// TwinCAT 3 PLC project Untitled1
// ProgramVersion: 3.1.4023.0
// libraries:
//   Tc2_MC2, * (Beckhoff Automation GmbH)
//   Tc2_Standard, * (Beckhoff Automation GmbH)
//   Tc2_System, * (Beckhoff Automation GmbH)
//   Tc2_Utilities, * (Beckhoff Automation GmbH)
//   Tc3_Module, * (Beckhoff Automation GmbH)
// project tree:
//   DUTs/ A21ToolStorage.TcDUT (not stored), Bundle.TcDUT (not stored), EOAT.TcDUT (not stored), Interval.TcDUT (not stored), ONE_BIT.TcDUT (not stored), PositionMaterials.TcDUT (not stored)
//   DUTs/Enums/ A21.TcDUT (not stored), Chipboard.TcDUT (not stored), Homing.TcDUT (not stored), SectionEnum.TcDUT (not stored), Surface.TcDUT (not stored), WoodBunk.TcDUT (not stored)
//   DUTs/Insertion/Drives/ AirPiston.TcPOU (not stored), ClearLinkMC.TcPOU, SimplePiston.TcPOU (not stored)
//   DUTs/Insertion/ Insertion.TcPOU, SuctionPad.TcDUT (not stored)
//   DUTs/Insertion/Prototypes/ FBA_Drive.TcPOU, I_ContinuousDrive.TcIO (not stored), I_Drive.TcIO, I_PositionalDrive.TcIO (not stored), I_EncodedDrive.TcIO (not stored)
//   DUTs/Machines/ KukaRobot.TcPOU, RobotA21.TcPOU, StrapMachine.TcPOU
//   DUTs/Material Holders/ SkidMagazine.TcPOU, MaterialHolder.TcPOU, WoodBunkTable.TcPOU
//   GVLs/ GVL.TcGVL (not stored), Hardware.TcGVL
//   / PlcTask.TcTTO
//   POUs/ MAIN.TcPOU
//   POUs/Module Calls/ CallHardwareModules.TcPOU, SetSuctions.TcPOU (not stored), SetupHardware.TcPOU
//   POUs/Utility/ BoolArrayToInteger.TcPOU, CEILING.TcPOU (not stored), IntegerBitAccess.TcPOU (not stored), IntegerToBoolArray.TcPOU (not stored), JoinStrings.TcPOU (not stored), WithinTolerance.TcPOU (not stored)
//   POUs/Utility/String Array/ AddToStringArray.TcPOU, RemoveElementFromStringArray.TcPOU (not stored), RemoveIndexFromStringArray.TcPOU (not stored), StringArrayCloseGaps.TcPOU (not stored)
// real-time tasks:
//   TASK PlcTask: cycle T#10ms, priority 20, ADS port 350
// I/O:
//   DEVICE Device 1 (EtherCAT), AmsNetId 5.131.216.41.2.1
//     EK1200 [EK1200-5000 EtherCAT Power supply (2A E-Bus)]
//       IPC_O [EL2809 16Ch. Dig. Output 24V, 0.5A]
//       JUNC_A21 [EK1122 2 port EtherCAT junction]
//         C4 [EK1100 EtherCAT Coupler (2A E-Bus)]
//           C4_I1 [EL1809 16Ch. Dig. Input 24V, 3ms]
//           C4_O2 [EL2809 16Ch. Dig. Output 24V, 0.5A]
//           C4_O3 [EL2809 16Ch. Dig. Output 24V, 0.5A]
//           BRIDGE_ROBOT1 [EL6695 EtherCAT Bridge terminal (Primary)]
//           Term 14 (EL9011) [EL9011 End Terminal]
//         SB01 [EP1809-0021 16 Ch. Dig. Input 24V, 3ms, M8]
//         SB05 [EP1008-0001 8 Ch. Dig. Input 24V, 3ms, M8]
//         SB04 [EP1809-0021 16 Ch. Dig. Input 24V, 3ms, M8]
//         SB03 [EP1008-0001 8 Ch. Dig. Input 24V, 3ms, M8]
//         C1 [EK1100 EtherCAT Coupler (2A E-Bus)]
//           C1_I1 [EL1809 16Ch. Dig. Input 24V, 3ms]
//           C1_O2 [EL2809 16Ch. Dig. Output 24V, 0.5A]
//           BRIDGE_ROBOT2 [EL6695 EtherCAT Bridge terminal (Primary)]
//           Term 13 (EL9011) [EL9011 End Terminal]
//         SB02 [EP1809-0021 16 Ch. Dig. Input 24V, 3ms, M8]
//         SB07 [EP1008-0001 8 Ch. Dig. Input 24V, 3ms, M8]
//         SB06 [EP1008-0001 8 Ch. Dig. Input 24V, 3ms, M8]
// variable links:
//   Untitled1/Untitled1 Instance <-> Device 1 (EtherCAT)/EK1200/JUNC_A21/C1/BRIDGE_ROBOT2
//     PlcTask Inputs/Hardware.robotRight.inputs[{2..20}] <-> IO Inputs/In_{2..20}  (19 links)
//     PlcTask Inputs/Hardware.robotRight.inputs[1] <-> IO Inputs/In
//     PlcTask Outputs/Hardware.robotRight.outputs[{2..50}] <-> IO Outputs/Out_{2..50}  (49 links)
//     PlcTask Outputs/Hardware.robotRight.outputs[1] <-> IO Outputs/Out
//   Untitled1/Untitled1 Instance <-> Device 1 (EtherCAT)/EK1200/JUNC_A21/C1/C1_I1
//     PlcTask Inputs/Hardware.strapper.done <-> Channel 4/Input
//     PlcTask Inputs/Hardware.strapper.error <-> Channel 1/Input
//     PlcTask Inputs/Hardware.strapper.home <-> Channel 5/Input
//     PlcTask Inputs/Hardware.strapper.ready <-> Channel 2/Input
//   Untitled1/Untitled1 Instance <-> Device 1 (EtherCAT)/EK1200/JUNC_A21/C1/C1_O2
//     PlcTask Outputs/Hardware.strapper.enable <-> Channel 2/Output
//     PlcTask Outputs/Hardware.strapper.execute <-> Channel 1/Output
//     PlcTask Outputs/Hardware.strapper.reset <-> Channel 3/Output
//   Untitled1/Untitled1 Instance <-> Device 1 (EtherCAT)/EK1200/JUNC_A21/C4/BRIDGE_ROBOT1
//     PlcTask Inputs/Hardware.robotLeft.inputs[{2..20}] <-> IO Inputs/In_{2..20}  (19 links)
//     PlcTask Inputs/Hardware.robotLeft.inputs[1] <-> IO Inputs/In
//     PlcTask Outputs/Hardware.robotLeft.outputs[{2..50}] <-> IO Outputs/Out_{2..50}  (49 links)
//     PlcTask Outputs/Hardware.robotLeft.outputs[1] <-> IO Outputs/Out
//   Untitled1/Untitled1 Instance <-> Device 1 (EtherCAT)/EK1200/JUNC_A21/C4/C4_I1
//     PlcTask Inputs/Hardware.topSuction[1].occupied <-> Channel 9/Input
//     PlcTask Inputs/Hardware.topSuction[2].occupied <-> Channel 10/Input
//     PlcTask Inputs/Hardware.topSuction[3].occupied <-> Channel 11/Input
//     PlcTask Inputs/Hardware.verticalDriveLeft.home <-> Channel 3/Input
//     PlcTask Inputs/Hardware.verticalDriveLeft.innerLimit <-> Channel 2/Input
//     PlcTask Inputs/Hardware.verticalDriveLeft.outerLimit <-> Channel 1/Input
//     PlcTask Inputs/Hardware.verticalDriveRight.home <-> Channel 7/Input
//     PlcTask Inputs/Hardware.verticalDriveRight.innerLimit <-> Channel 6/Input
//     PlcTask Inputs/Hardware.verticalDriveRight.outerLimit <-> Channel 5/Input
//   Untitled1/Untitled1 Instance <-> Device 1 (EtherCAT)/EK1200/JUNC_A21/C4/C4_O2
//     PlcTask Outputs/Hardware.horizontalDriveLeft.valveExtend <-> Channel 5/Output
//     PlcTask Outputs/Hardware.horizontalDriveLeft.valveRetract <-> Channel 6/Output
//     PlcTask Outputs/Hardware.horizontalDriveRight.valveExtend <-> Channel 15/Output
//     PlcTask Outputs/Hardware.horizontalDriveRight.valveRetract <-> Channel 16/Output
//     PlcTask Outputs/Hardware.leftSuction[{1..4}].enable <-> Channel {7..10}/Output  (4 links)
//     PlcTask Outputs/Hardware.verticalDriveLeft.brakeRelease <-> Channel 4/Output
//     PlcTask Outputs/Hardware.verticalDriveRight.brakeRelease <-> Channel 14/Output
//   Untitled1/Untitled1 Instance <-> Device 1 (EtherCAT)/EK1200/JUNC_A21/C4/C4_O3
//     PlcTask Outputs/Hardware.bottomSuction[1].enable <-> Channel 7/Output
//     PlcTask Outputs/Hardware.bottomSuction[2].enable <-> Channel 8/Output
//     PlcTask Outputs/Hardware.pistonBottom.pistonExtend <-> Channel 5/Output
//     PlcTask Outputs/Hardware.pistonBottom.pistonRetract <-> Channel 6/Output
//     PlcTask Outputs/Hardware.rightSuction[{1..4}].enable <-> Channel {1..4}/Output  (4 links)
//     PlcTask Outputs/Hardware.topSuction[1].enable <-> Channel 9/Output
//     PlcTask Outputs/Hardware.topSuction[2].enable <-> Channel 10/Output
//     PlcTask Outputs/Hardware.topSuction[3].enable <-> Channel 11/Output
//   Untitled1/Untitled1 Instance <-> Device 1 (EtherCAT)/EK1200/JUNC_A21/SB01
//     PlcTask Inputs/Hardware.horizontalDriveLeft.home <-> Channel 11/Input
//     PlcTask Inputs/Hardware.horizontalDriveLeft.innerLimit <-> Channel 12/Input
//     PlcTask Inputs/Hardware.leftSuction[{1..4}].occupied <-> Channel {13..16}/Input  (4 links)
//     PlcTask Inputs/Hardware.stagingTableLeft.occupied[{1..10}] <-> Channel {1..10}/Input  (10 links)
//   Untitled1/Untitled1 Instance <-> Device 1 (EtherCAT)/EK1200/JUNC_A21/SB02
//     PlcTask Inputs/Hardware.horizontalDriveRight.home <-> Channel 11/Input
//     PlcTask Inputs/Hardware.horizontalDriveRight.innerLimit <-> Channel 12/Input
//     PlcTask Inputs/Hardware.rightSuction[{1..4}].occupied <-> Channel {13..16}/Input  (4 links)
//     PlcTask Inputs/Hardware.stagingTableRight.occupied[{1..10}] <-> Channel {1..10}/Input  (10 links)
//   Untitled1/Untitled1 Instance <-> Device 1 (EtherCAT)/EK1200/JUNC_A21/SB05
//     PlcTask Inputs/Hardware.magazineLeft.inPosition1 <-> Channel 1/Input
//     PlcTask Inputs/Hardware.magazineLeft.inPosition2 <-> Channel 2/Input
//     PlcTask Inputs/Hardware.skidLeft.inPosition1 <-> Channel 3/Input
//     PlcTask Inputs/Hardware.skidLeft.inPosition2 <-> Channel 4/Input
//   Untitled1/Untitled1 Instance <-> Device 1 (EtherCAT)/EK1200/JUNC_A21/SB06
//     PlcTask Inputs/Hardware.magazineRight.inPosition1 <-> Channel 1/Input
//     PlcTask Inputs/Hardware.magazineRight.inPosition2 <-> Channel 2/Input
//     PlcTask Inputs/Hardware.skidRight.inPosition1 <-> Channel 3/Input
//     PlcTask Inputs/Hardware.skidRight.inPosition2 <-> Channel 4/Input
//   Untitled1/Untitled1 Instance <-> Device 1 (EtherCAT)/EK1200/JUNC_A21/SB07
//     PlcTask Inputs/Hardware.bottomSuction[1].occupied <-> Channel 6/Input
//     PlcTask Inputs/Hardware.bottomSuction[2].occupied <-> Channel 7/Input
//     PlcTask Inputs/Hardware.pistonBottom.extended <-> Channel 5/Input
//     PlcTask Inputs/Hardware.pistonBottom.retracted <-> Channel 4/Input

CONFIGURATION Untitled1
    RESOURCE PLC ON TwinCAT3
        TASK PlcTask(INTERVAL := T#10ms, PRIORITY := 20);
        PROGRAM MAIN WITH PlcTask : MAIN;
    END_RESOURCE
END_CONFIGURATION

// ---- GVLs/Hardware.TcGVL
//{attribute 'qualified_only'}
VAR_GLOBAL
	robotLeft, robotRight : RobotA21;
	toolStorageLeft, toolStorageRight : A21ToolStorage;
	
	skidLeft, skidRight : SkidMagazine;
	
	stagingTableLeft, stagingTableRight : WoodBunkTable;
	magazineLeft, magazineRight : SkidMagazine;
	
	strapper : StrapMachine;
	
	horizontalDriveLeft, horizontalDriveRight : AirPiston;
	verticalDriveLeft, verticalDriveRight : ClearLinkMC;
	pistonBottom : SimplePiston;
	
	topSuction : ARRAY[1..3] OF SuctionPad;
	leftSuction : ARRAY[1..4] OF SuctionPad;
	rightSuction : ARRAY[1..4] OF SuctionPad; 
	bottomSuction : ARRAY[1..2] OF SuctionPad;
END_VAR

// ---- DUTs/Insertion/Prototypes/I_Drive.TcIO
INTERFACE I_Drive

PROPERTY ABSTRACT AtHome : BOOL
GET
END_GET
END_PROPERTY

PROPERTY ABSTRACT AtInnerLimit : BOOL
GET
END_GET
END_PROPERTY

PROPERTY ABSTRACT AtOuterLimit : BOOL
GET
END_GET
END_PROPERTY

PROPERTY ABSTRACT Busy : BOOL
GET
END_GET
END_PROPERTY

PROPERTY ABSTRACT Contact : BOOL
GET
END_GET
END_PROPERTY

PROPERTY ABSTRACT Error : BOOL
GET
END_GET
END_PROPERTY

PROPERTY ABSTRACT HomeSet : BOOL
GET
END_GET
END_PROPERTY

METHOD ABSTRACT homingSequence : BOOL
VAR_INPUT
END_VAR
END_METHOD

METHOD ABSTRACT stop : BOOL
VAR_INPUT
END_VAR
END_METHOD

END_INTERFACE

// ---- POUs/MAIN.TcPOU
PROGRAM MAIN
VAR
	execute : BOOL;
	stop : BOOL;
	generalError : BOOL;
	failLeft, failRight : BOOL;
	
	manualStep : BOOL := TRUE;
	manualSuction : BOOL := FALSE;
END_VAR
VAR //local types
	woodBunkArr : ARRAY[0..GVL.maxPairs] OF PositionMaterials;
	
	stagingTemplateLeft, stagingTemplateRight AT %M* : WoodBunkTable; //declaration with %M* overwrites addresses of local attributes
	stagingArrayLeft, stagingArrayRight : ARRAY[0..GVL.maxPairs*2] OF STRING;
	insertionLeft, insertionRight : Insertion;
END_VAR
VAR //for testing, to be removed when replaced with pressure sensors
	latchLeft, latchRight : BOOL; //prevents SMC sliders from overshooting the inner limit sensor
	
	suctionEnableTop : BOOL;
	suctionEnableLeft : BOOL;
	suctionEnableRight : BOOL;
	suctionEnableBottom : BOOL;
	
	done : BOOL;
	
	demoPairWB : PositionMaterials := (
		position := 0,
		top := 'WDS20',
		left := 'WDS20',
		right := 'WDS20',
		bottom := 'WDS14');
		
	demoPairCIP : PositionMaterials := (
		position := 0,
		top := 'CIP54',
		bottom := 'CIP18');
	
	demoHeight : REAL := 600; //mm
END_VAR
VAR
	robotLeftOutputs, robotRightOutputs : ARRAY[1..11] OF INT;
	
	insertionMaterials : ARRAY[Surface.TOP..Surface.BOTTOM] OF STRING;
	//robotLeftMaterial, robotRightMaterial : STRING;
	
	topSuctionDelay : TON;
	
	step : (IDLE, LOAD_CIP, STAGING, LOAD_WB, PUSH, STRAP, RELEASE, COMPLETE := 1050);
	
	//these 2 ints should replace the 4 ints after
	commandSet : INT;
	commandStepLeft, commandStepRight : INT;
	
	loadSet : INT;
	loadStepLeft, loadStepRight : INT;
	
	stageSet : INT;	
	stageStepLeft, stageStepRight : INT;
	iSlotLeft, iSlotRight : INT(1..10);
END_VAR
VAR //CONSTANT
	sectionID : SectionEnum := SectionEnum.CHIPBOARD;
	idleRobotOutput : ARRAY[1..11] OF INT;
END_VAR

SetupHardware();
CallHardwareModules();
callLocalModules();

woodBunkArr[0] := demoPairWB;

IF stop THEN //may need to turn off suction
	insertionLeft.stop();
	insertionRight.stop();
	pistonBottom.stop();
	
	robotLeft.clearCommand();
	robotRight.clearCommand();
	RETURN;
END_IF


IF NOT (insertionLeft.screw.HomeSet AND insertionRight.screw.HomeSet) THEN
	insertionLeft.homingSequence();
	insertionRight.homingSequence();
	pistonBottom.retract();
	RETURN;
END_IF


CASE step OF
	IDLE:
		IF execute THEN
			execute := FALSE;
			suctionEnableTop := suctionEnableLeft := suctionEnableRight := suctionEnableBottom := FALSE;
			step := STAGING;
		END_IF
		
		SetSuctions(topSuction, suctionEnableTop);
		SetSuctions(leftSuction, suctionEnableLeft);
		SetSuctions(rightSuction, suctionEnableRight);
		SetSuctions(bottomSuction, suctionEnableBottom);
		
	LOAD_CIP:
		IF NOT done THEN
			done := loadCIP(pair:= demoPairWB, error => generalError);
		END_IF
		
		IF
			(manualStep AND_THEN execute) OR
			(NOT manualStep AND_THEN done)
		THEN
			done := FALSE;
			execute := FALSE;
			
			step := STAGING;
		END_IF
		
	STAGING:
		IF NOT done THEN
			done := stage(error => generalError);
		END_IF
		
		IF
			(manualStep AND_THEN execute) OR
			(NOT manualStep AND_THEN done)
		THEN
			execute := FALSE;
			done := FALSE;
			step := LOAD_WB;
		END_IF
	
	LOAD_WB:
		IF NOT done THEN
			done := loadWB(pair := demoPairWB, error => generalError);
		END_IF
		
		IF manualSuction THEN
			SetSuctions(topSuction, suctionEnableTop);
			SetSuctions(leftSuction, suctionEnableLeft);
			SetSuctions(rightSuction, suctionEnableRight);
			SetSuctions(bottomSuction, suctionEnableBottom);
		END_IF
		
		IF
			(manualStep AND_THEN execute) OR
			(NOT manualStep AND_THEN done)
		THEN
			done := FALSE;
			suctionEnableTop := suctionEnableLeft := suctionEnableRight := suctionEnableBottom := FALSE;
			execute := FALSE;
			
			step := PUSH;
		END_IF
		
	PUSH:
		(*
		IF 
			insertionLeft.sliderPos <> demoHeight/2 //OR 
			//insertionRight.sliderPos <> demoHeight/2 //OR 
			//NOT insertionBottom.contact
		THEN
			insertionLeft.slideAbsolute(demoHeight/2);
			//insertionRight.slideAbsolute(demoHeight/2);
			RETURN;
		END_IF
		*)
		
		IF insertionLeft.screw.AtInnerLimit THEN
			latchLeft := TRUE;
		ELSIF NOT latchLeft THEN
			insertionLeft.press();
		END_IF
		
		IF insertionRight.screw.AtInnerLimit THEN
			latchRight := TRUE;
		ELSIF NOT latchRight THEN
			insertionRight.press();
		END_IF
		pistonBottom.extend();
		
		IF
			(manualStep AND_THEN execute) OR
			(latchLeft AND latchRight (*AND insertionBottom.extended*))
		THEN
			latchLeft := latchRight := FALSE;
			execute := FALSE;
			step := STRAP;
		END_IF
		
	STRAP:
		topSuctionDelay(IN:= , PT:= T#1S, Q=> , ET=> );
		
		strapper.bEnable := TRUE;
		IF strapper.done THEN
			topSuctionDelay.IN := FALSE;
			step := RELEASE;
			RETURN;
		END_IF
		
		IF topSuctionDelay.Q THEN
			SetSuctions(topSuction, FALSE);
			SetSuctions(leftSuction, FALSE);
			SetSuctions(rightSuction, FALSE);
			SetSuctions(bottomSuction, FALSE);
		ELSIF strapper.atBundleLevel THEN
			topSuctionDelay.IN := TRUE;
		END_IF
		
		IF strapper.ready THEN
			strapper.strap();
		END_IF
		
		IF execute THEN
			topSuctionDelay.IN := FALSE;
			execute := FALSE;
			step := RELEASE;
		END_IF
		
	RELEASE: //release command		
		//insertionLeft.slideAbsolute(0);
		//insertionRight.slideAbsolute(0);
		
		insertionLeft.release();
		insertionRight.release();
		pistonBottom.retract();
		
		IF 
			(insertionLeft.screw.AtHome AND insertionRight.screw.AtHome AND pistonBottom.retracted) OR
			execute
		THEN
			execute := FALSE;
			step := COMPLETE;
		END_IF
	
	COMPLETE:
		//reset everything
		step := IDLE;
		
END_CASE

CallHardwareModules(); //end program with hardware call

METHOD callLocalModules : BOOL
stagingTemplateLeft();
stagingTemplateRight();

insertionLeft(
	enable:= TRUE, 
	slider:= verticalDriveLeft, 
	screw:= horizontalDriveLeft, 
	contact=> , 
	softContact=> , 
	busy=> , 
	error=> , 
	home=> , 
	homingComplete=> , 
	sliderPos=> );
	
insertionRight(
	enable:= TRUE, 
	slider:= verticalDriveRight, 
	screw:= horizontalDriveRight,  
	contact=> , 
	softContact=> , 
	busy=> , 
	error=> , 
	home=> , 
	homingComplete=> , 
	sliderPos=> );
END_METHOD

METHOD changeRobotsEOAT : BOOL
VAR_IN_OUT
	robot : RobotA21;
END_VAR
VAR_INPUT
	targetTool : SectionEnum;
END_VAR
IF robotLeft.tool <> targetTool THEN
	MEMSET(ADR(robotLeftOutputs), 0, SIZEOF(robotLeftOutputs));
	
	CASE targetTool OF
		SectionEnum.CHIPBOARD: robotLeftOutputs[1] := A21.TOOL_CHANGE_CHIPBOARD;
		SectionEnum.WOOD_BUNK: robotLeftOutputs[1] := A21.TOOL_CHANGE_BUNK;
	END_CASE
	
	robotLeft.setCommand(robotLeftOutputs);
END_IF

IF robotRight.tool <> targetTool THEN
	MEMSET(ADR(robotRightOutputs), 0, SIZEOF(robotRightOutputs));
	
	CASE targetTool OF
		SectionEnum.CHIPBOARD: robotLeftOutputs[1] := A21.TOOL_CHANGE_CHIPBOARD;
		SectionEnum.WOOD_BUNK: robotLeftOutputs[1] := A21.TOOL_CHANGE_BUNK;
	END_CASE
	
	robotRight.setCommand(robotRightOutputs);
END_IF

changeRobotsEOAT := robot.tool = targetTool;

(*
IF robot.gripper.id <> targetTool THEN
	CASE targetTool OF
		SectionEnum.CHIPBOARD:	robot.setGroup(group := 1, value := A21.TOOL_CHANGE_CHIPBOARD);
		SectionEnum.WOOD_BUNK:	robot.setGroup(group := 1, value := A21.TOOL_CHANGE_BUNK);
	END_CASE
END_IF

changeRobotsEOAT := robot.gripper.id = targetTool;
*)
END_METHOD

METHOD createStagingArrayLeft : BOOL
VAR
	remainingMaterial : STRING;
	splitMaterial : STRING;
	
	i : INT;
END_VAR
FOR i:=0 TO GVL.maxPairs BY 1 DO
	remainingMaterial := woodBunkArr[i].top;
	WHILE FIND(remainingMaterial, '_') > 0 DO
		splitCombinedMaterials(remainingMaterial, splitMaterial);
		IF splitMaterial <> '' THEN
			AddToStringArray(arr := stagingArrayLeft, newString := splitMaterial, numElements => , nextIndex => );
		END_IF
	END_WHILE
	
	IF remainingMaterial <> '' THEN
		AddToStringArray(arr := stagingArrayLeft, newString := remainingMaterial, numElements => , nextIndex => );
	END_IF
	
	
	remainingMaterial := woodBunkArr[i].left;
	WHILE FIND(remainingMaterial, '_') > 0 DO
		splitCombinedMaterials(remainingMaterial, splitMaterial);
		IF splitMaterial <> '' THEN
			AddToStringArray(arr := stagingArrayLeft, newString := splitMaterial, numElements => , nextIndex => );
		END_IF
	END_WHILE
	
	IF remainingMaterial <> '' THEN
		AddToStringArray(arr := stagingArrayLeft, newString := remainingMaterial, numElements => , nextIndex => );
	END_IF
END_FOR
END_METHOD

METHOD createStagingArrayRight : BOOL
VAR
	remainingMaterial : STRING;
	splitMaterial : STRING;
	
	i : INT;
END_VAR
FOR i:=0 TO GVL.maxPairs*2 BY 1 DO
	remainingMaterial := woodBunkArr[i].bottom;
	WHILE FIND(remainingMaterial, '_') > 0 DO
		splitCombinedMaterials(remainingMaterial, splitMaterial);
		IF splitMaterial <> '' THEN
			AddToStringArray(arr := stagingArrayRight, newString := splitMaterial, numElements => , nextIndex => );
		END_IF
	END_WHILE
	
	IF remainingMaterial <> '' THEN
		AddToStringArray(arr := stagingArrayRight, newString := remainingMaterial, numElements => , nextIndex => );
	END_IF
	
	
	
	remainingMaterial := woodBunkArr[i].right;
	WHILE FIND(remainingMaterial, '_') > 0 DO
		splitCombinedMaterials(remainingMaterial, splitMaterial);
		IF splitMaterial <> '' THEN
			AddToStringArray(arr := stagingArrayRight, newString := splitMaterial, numElements => , nextIndex => );
		END_IF
	END_WHILE
	
	IF remainingMaterial <> '' THEN
		AddToStringArray(arr := stagingArrayRight, newString := remainingMaterial, numElements => , nextIndex => );
	END_IF
END_FOR
END_METHOD

METHOD PROTECTED generateStagingTemplate : BOOL
VAR
	remainingMaterial : STRING;
	splitMaterial : STRING;
	
	i : INT;
END_VAR
VAR_STAT
	temp : INT;
END_VAR
createStagingArrayLeft();
createStagingArrayRight();

//AddToStringArray(arr := stagingArrayLeft, newString := 'WDB20', numElements =>, nextIndex => );

(*
iterate through all pairs and autofill the template
replace succesfully autofilled materials with empty string

when staging needs to be performed a 2nd time, autofilling empty strings is always unsuccessful
*)
FOR i:=0 TO GVL.maxPairs*2 BY 1 DO
	IF stagingTemplateLeft.autofill(materialID := stagingArrayLeft[i]) THEN
		stagingArrayLeft[i] := '';
	END_IF
	
	IF stagingTemplateRight.autofill(materialID := stagingArrayRight[i]) THEN
		stagingArrayRight[i] := '';
	END_IF
END_FOR

(*
stagingTemplateLeft.autofill(demoPairWB.top);
stagingTemplateLeft.autofill(demoPairWB.left);

stagingTemplateRight.autofill(demoPairWB.right);
stagingTemplateRight.autofill(demoPairWB.bottom);
*)

generateStagingTemplate := TRUE;
END_METHOD

METHOD loadCIP : BOOL
VAR_INPUT
	pair : REFERENCE TO PositionMaterials;
END_VAR
VAR_OUTPUT
	error : BOOL;
END_VAR
sectionID := SectionEnum.CHIPBOARD;

IF NOT robotLeft.operational AND NOT robotLeft.operational THEN //robots not operational
	error := TRUE;
	RETURN;
END_IF

IF NOT (robotLeft.reserve(sectionID) AND robotRight.reserve(sectionID)) THEN //robots not reserved
	RETURN;
END_IF

IF NOT (robotLeft.tool = sectionID AND robotRight.tool = sectionID) THEN //robots have wrong tool
	changeRobotsEOAT(robot := robotLeft, targetTool := sectionID); //wait for robots to finish changing tools
	changeRobotsEOAT(robot := robotRight, targetTool := sectionID);
	RETURN;
END_IF
//robots ok

CASE loadSet OF
	0: //demo only - only top chipboard loaded by left robot
		IF 
			loadingSequenceCIP(
				robot:= robotLeft, 
				command:= robotLeftOutputs, 
				storage:= skidLeft, 
				loadStep:= loadStepLeft, 
				surfaceID:= Surface.TOP,
				material:= pair.top, 
				fail=> )
		THEN
			loadStepLeft := loadStepRight := 0;
			loadSet := 10;
		END_IF
		
	10: //recovery
		IF robotLeft.operational AND NOT robotRight.operational THEN //left ok, right fail
			IF //load bottom using left robot
				loadingSequenceCIP(
					robot:= robotLeft, 
					command:= robotLeftOutputs, 
					storage:= skidLeft, 
					loadStep:= loadStepLeft, 
					surfaceID:= Surface.BOTTOM,
					material:= pair.top, 
					fail=> ) //load bottom with left robot
			THEN
				loadSet := COMPLETE;
			END_IF
			
		ELSIF NOT robotLeft.operational AND robotRight.operational THEN //left fail, right ok
			IF //load top using right robot
				loadingSequenceCIP(
					robot:= robotRight, 
					command:= robotRightOutputs, 
					storage:= skidRight, 
					loadStep:= loadStepRight, 
					surfaceID:= Surface.TOP,
					material:= pair.bottom, 
					fail=> ) //load top with right robot
			THEN
				loadSet := COMPLETE;
			END_IF
			
		END_IF
		
	COMPLETE:
		loadSet := 0;
		loadStepLeft := loadStepRight := 0;
		
		robotLeft.release(sectionID);
		robotRight.release(sectionID);
		
		loadCIP := TRUE;
END_CASE
END_METHOD

METHOD loadingSequenceCIP : BOOL
VAR_IN_OUT
	robot : RobotA21;
	command : ARRAY[1..11] OF INT;
	storage : MaterialHolder;
	loadStep : INT;
END_VAR
VAR_INPUT
	surfaceID : Surface;
	material : STRING;
END_VAR
VAR_OUTPUT
	fail : BOOL;
END_VAR
VAR
	slot : INT;
END_VAR
IF material = '' THEN
	loadingSequenceCIP := TRUE;
	RETURN;
END_IF

CASE loadStep OF
	0:
		IF NOT storage.findSlot(materialID := material, atSlot => slot) THEN
			fail := TRUE;
			RETURN;
		END_IF
		
		MEMSET(ADR(command), 0, SIZEOF(command));
		command[1] := A21.GET_CHIPBOARD_FROM_SKID;
		command[2] := slot;
		
		IF surfaceID = Surface.BOTTOM THEN
			//lower conveyor
		END_IF
		
		CASE surfaceID OF
			Surface.TOP:
				IF robot.setCommand(command) THEN
					loadStep := 10;
				END_IF
				
			Surface.BOTTOM:
				//lower conveyor
				IF robot.setCommand(command) (*AND conveyor lowered*) THEN
					loadStep := 10;
				END_IF
			
		END_CASE
		
	10:
		MEMSET(ADR(command), 0, SIZEOF(command));
		CASE surfaceID OF
			Surface.TOP: 					command[1] := A21.PLACE_CHIPBOARD_TO_TOP;
			Surface.BOTTOM: 				command[1] := A21.PLACE_CHIPBOARD_TO_BOTTOM;
		END_CASE
		command[2] := slot;
		
		IF robot.setCommand(command) THEN
			loadStep := 10;
		END_IF
		
	COMPLETE:
		robot.release(sectionID);
		loadingSequenceCIP := TRUE;
		
END_CASE
END_METHOD

METHOD loadingSequenceWB : BOOL
VAR_IN_OUT
	robot : RobotA21;
	//carryMaterial : STRING;
	table : WoodBunkTable;
	suctions : ARRAY[*] OF SuctionPad;
	loadStep : INT;
	slot : INT(1..10);
END_VAR
VAR_INPUT
	surfaceID : Surface;
	material : STRING;
END_VAR
VAR_OUTPUT
	fail : BOOL;
END_VAR
VAR
	i : DINT;
END_VAR
VAR_STAT
	tempSlot : INT;
END_VAR
IF material = '' THEN
	loadingSequenceWB := TRUE;
	RETURN;
END_IF

CASE loadStep OF
	0: //wait for robot
		robot.clearCommand();
		
		IF robot.Ready THEN
			loadStep := 10;
		END_IF
		
	10: //grab from table
		IF NOT table.findSlot(materialID := material, atSlot => slot) (*AND slot < 1*) THEN	//cannot find material on table	
			
			fail := TRUE;
			RETURN;
		END_IF
		tempSlot := slot;
		IF NOT table.occupied[slot] AND robot.suspendedMaterial = '' THEN //move from table to robot gripper
			robot.CarryMaterial := table.slots[slot];
			table.remove(i := slot, materialID => );
		END_IF
		
		IF robot.Done THEN
			loadStep := COMPLETE;
			RETURN;
		ELSIF robot.materialAtHoldingPosition >= 1 AND robot.materialAtHoldingPosition <= 8 THEN
			loadStep := 20;
			RETURN;
		END_IF
		
		CASE surfaceID OF
			Surface.TOP: 					robot.setGroup(group := 1, value := A21.LOAD_BUNK_TO_TOP); 
			Surface.LEFT, Surface.RIGHT: 	robot.setGroup(group := 1, value := A21.LOAD_BUNK_TO_SIDE);
			Surface.BOTTOM: 				robot.setGroup(group := 1, value := A21.LOAD_BUNK_TO_BOTTOM);
		END_CASE
		robot.setGroup(group := 2, value := slot); 
			
	20: //place to insertion
		IF robotLeft.Done THEN
			loadStep := COMPLETE;
			RETURN;
		END_IF
		
		robot.setGroup(group := 9, value := robot.inputs[5]);
		
		IF robot.materialAtHoldingPosition > 0 AND robot.CarryMaterial <> '' THEN //move from gripper to insertion
			IF insertionMaterials[surfaceID] = '' THEN //transfer to insertion as is
				insertionMaterials[surfaceID] := robot.suspendedMaterial;
			ELSE //join with existing material using underscore _
				insertionMaterials[surfaceID] := JoinStrings(insertionMaterials[surfaceID], robot.suspendedMaterial, '_');
			END_IF
			robot.CarryMaterial := '';
		END_IF
		
		CASE surfaceID OF
			Surface.TOP, Surface.BOTTOM:
				SetSuctions(suctions, TRUE (*robot.materialAtHoldingPosition = 1 OR robot.materialAtHoldingPosition = 4*));
				
			Surface.LEFT, Surface.RIGHT:
				SetSuctions(suctions, TRUE (*robot.materialAtHoldingPosition = 2 OR robot.materialAtHoldingPosition = 3*));
				(*
				FOR i:=LOWER_BOUND(suctions, 1) TO UPPER_BOUND(suctions, 1) BY 1 DO
					
					IF i < UPPER_BOUND(suctions, 1)/2 THEN
						suctions[i].enable := robot.materialAtHoldingPosition = 2; //enable upper half suctions
					ELSE
						suctions[i].enable := robot.materialAtHoldingPosition = 3; //enable lower half suctions
					END_IF

				END_FOR
				*)
		END_CASE
	
	COMPLETE:
		robot.clearCommand();
		loadingSequenceWB := TRUE;
		
END_CASE
END_METHOD

METHOD loadingSequenceWB_old : BOOL
VAR_IN_OUT
	robot : RobotA21;
	commands : ARRAY[1..11] OF INT;
	carryMaterial : STRING;
	table : WoodBunkTable;
	suctions : ARRAY[*] OF SuctionPad;
	loadStep : INT;
	slot : INT(1..10);
END_VAR
VAR_INPUT
	surfaceID : Surface;
	material : STRING;
END_VAR
VAR_OUTPUT
	fail : BOOL;
END_VAR
VAR
	i : DINT;
END_VAR
IF material = '' THEN
	loadingSequenceWB_old := TRUE;
	RETURN;
END_IF

CASE loadStep OF
	0: //wait for robot
		IF robot.Ready THEN
			loadStep := 10;
		END_IF
		
	10: //grab from table
		IF NOT table.findSlot(materialID := material, atSlot => slot) (*AND slot < 1*) THEN	//cannot find material on table	
			fail := TRUE;
			RETURN;
		END_IF
		
		IF NOT table.occupied[slot] AND carryMaterial = '' THEN //move from table to robot gripper
			table.remove(i := slot, materialID => carryMaterial);
		END_IF
		
		IF robot.inputs[5] > 0 THEN
			loadStep := 20;
			RETURN;
		END_IF		
		
		MEMSET(ADR(commands), 0, SIZEOF(commands));
		CASE surfaceID OF
			Surface.TOP: 					commands[1] := A21.LOAD_BUNK_TO_TOP;
			Surface.LEFT, Surface.RIGHT: 	commands[1] := A21.LOAD_BUNK_TO_SIDE;
			Surface.BOTTOM: 				commands[1] := A21.LOAD_BUNK_TO_BOTTOM;
		END_CASE
		commands[2] := slot;
		robot.setCommand(commands);
			
	20: //place to insertion
		IF robotLeft.Done THEN
			loadStep := COMPLETE;
			RETURN;
		END_IF
		
		robot.setCommand(commands);
		robot.setGroup(group := 9, value := robot.inputs[5]);
		
		IF robot.inputs[5] > 0 THEN //move from gripper to insertion
			IF insertionMaterials[surfaceID] = '' THEN //transfer to insertion as is
				insertionMaterials[surfaceID] := carryMaterial;
			ELSE //join with existing material using underscore _
				insertionMaterials[surfaceID] := CONCAT(insertionMaterials[surfaceID], '_');
				insertionMaterials[surfaceID] := CONCAT(insertionMaterials[surfaceID], carryMaterial);
			END_IF
			carryMaterial := '';
		END_IF
		
		CASE surfaceID OF
			Surface.TOP, Surface.BOTTOM:
				SetSuctions(suctions, robot.inputs[5] = 1);
				
			Surface.LEFT, Surface.RIGHT:
				FOR i:=LOWER_BOUND(suctions, 1) TO UPPER_BOUND(suctions, 1) BY 1 DO
					
					IF i < UPPER_BOUND(suctions, 1)/2 THEN
						suctions[i].enable := robot.inputs[5] = 2; //enable upper half suctions
					ELSE
						suctions[i].enable := robot.inputs[5] = 3; //enable lower half suctions
					END_IF

				END_FOR
				(*
				suctions[1].enable := robot.inputs[5] = 2;
				suctions[2].enable := robot.inputs[5] = 2;
				
				suctions[3].enable := robot.inputs[5] = 3;
				suctions[4].enable := robot.inputs[5] = 3;
				*)
		END_CASE
		(*
		CASE robot.inputs[5] OF
			1, 4: //top/bottom insertions - enable all suctions
				SetSuctions(suctions, TRUE);
				
			2: //side insertion - enable upper half suctions
				suctions[1].enable := TRUE;
				suctions[2].enable := TRUE;
			
			3: //side insertion - enable lower half suctions
				suctions[3].enable := TRUE;
				suctions[4].enable := TRUE;
			
		END_CASE
		*)
	
	COMPLETE:
		robot.clearCommand();
		MEMSET(ADR(commands), 0, SIZEOF(commands));
		loadingSequenceWB_old := TRUE;
		
END_CASE
END_METHOD

METHOD loadingSequenceWB_simple : BOOL
VAR_IN_OUT
	robot : RobotA21;
	commands : ARRAY[1..11] OF INT;
	carryMaterial : STRING;
	table : WoodBunkTable;
	suctions : ARRAY[*] OF SuctionPad;
	loadStep : INT;
	slot : INT(1..10);
END_VAR
VAR_INPUT
	surfaceID : Surface;
	material : STRING;
END_VAR
VAR_OUTPUT
	fail : BOOL;
END_VAR
VAR
	i : DINT;
END_VAR
IF material = '' THEN
	loadingSequenceWB_simple := TRUE;
	RETURN;
END_IF

CASE loadStep OF
	0: //wait for robot
		IF robot.Ready THEN
			loadStep := 10;
		END_IF
		
	10: //grab from table
		IF NOT table.findSlot(materialID := material, atSlot => slot) (*AND slot < 1*) THEN	//cannot find material on table	
			fail := TRUE;
			RETURN;
		END_IF
		
		IF robotLeft.Done THEN
			loadStep := COMPLETE;
			RETURN;
		END_IF
		
		IF
			robot.inputs[5] > 0 AND  //robot is holding wood bunk at insertion position
			carryMaterial <> '' //robot gripper is carrying a wood bunk
		THEN
			//move from gripper to insertion
			IF insertionMaterials[surfaceID] = '' THEN //transfer to insertion as is
				insertionMaterials[surfaceID] := carryMaterial;
			ELSE //join with existing material using underscore _
				insertionMaterials[surfaceID] := CONCAT(insertionMaterials[surfaceID], '_');
				insertionMaterials[surfaceID] := CONCAT(insertionMaterials[surfaceID], carryMaterial);
			END_IF
			carryMaterial := '';
			
		ELSIF
			NOT table.occupied[slot] AND //table slot is vacant
			table.slots[slot] <> '' AND //table slot had a wood bunk on it
			carryMaterial <> '' //robot gripper is vacant
		THEN
			table.remove(i := slot, materialID => carryMaterial); //move from table to robot gripper
			
		END_IF		
		
		MEMSET(ADR(commands), 0, SIZEOF(commands));
		CASE surfaceID OF
			Surface.TOP: 					commands[1] := A21.LOAD_BUNK_TO_TOP;
			Surface.LEFT, Surface.RIGHT: 	commands[1] := A21.LOAD_BUNK_TO_SIDE;
			Surface.BOTTOM: 				commands[1] := A21.LOAD_BUNK_TO_BOTTOM;
		END_CASE
		commands[2] := slot;
		
		robot.setCommand(commands);
		robot.setGroup(group := 9, value := robot.inputs[5]);
		
		CASE surfaceID OF
			Surface.TOP, Surface.BOTTOM:
				SetSuctions(suctions, robot.inputs[5] = 1);
				
			Surface.LEFT, Surface.RIGHT:
				FOR i:=LOWER_BOUND(suctions, 1) TO UPPER_BOUND(suctions, 1) BY 1 DO
					
					IF i < UPPER_BOUND(suctions, 1)/2 THEN
						suctions[i].enable := robot.inputs[5] = 2; //enable upper half suctions
					ELSE
						suctions[i].enable := robot.inputs[5] = 3; //enable lower half suctions
					END_IF

				END_FOR
				(*
				//if the FOR loop does not work, use this
				suctions[1].enable := robot.inputs[5] = 2;
				suctions[2].enable := robot.inputs[5] = 2;
				
				suctions[3].enable := robot.inputs[5] = 3;
				suctions[4].enable := robot.inputs[5] = 3;
				*)
		END_CASE
		(*
		//if the above does not work, revert to this
		CASE robot.inputs[5] OF
			1, 4: //top/bottom insertions - enable all suctions
				SetSuctions(suctions, TRUE);
				
			2: //side insertion - enable upper half suctions
				suctions[1].enable := TRUE;
				suctions[2].enable := TRUE;
			
			3: //side insertion - enable lower half suctions
				suctions[3].enable := TRUE;
				suctions[4].enable := TRUE;
		END_CASE
		*)		
	
	COMPLETE:
		robot.clearCommand();
		MEMSET(ADR(commands), 0, SIZEOF(commands));
		loadingSequenceWB_simple := TRUE;
		
END_CASE
END_METHOD

METHOD PROTECTED loadWB : BOOL
VAR_INPUT
	pair : REFERENCE TO PositionMaterials;
END_VAR
VAR_OUTPUT
	error : BOOL;
END_VAR
VAR_STAT
	leftMaterial : STRING;
	rightMaterial : STRING;
END_VAR
sectionID := SectionEnum.WOOD_BUNK;

(*
IF NOT robotLeft.operational OR NOT robotLeft.operational THEN
	error := TRUE;
	RETURN;
END_IF
*)

IF robotLeft.error OR robotRight.error THEN
	error := TRUE;
	RETURN;
	
ELSIF NOT (robotLeft.reserve(sectionID) AND robotRight.reserve(sectionID)) THEN //loading requires both robots be reserved together
	RETURN;
	
ELSIF
	(robotLeft.tool <> sectionID AND_THEN NOT changeRobotsEOAT(robot := robotLeft, targetTool := sectionID)) OR
	(robotRight.tool <> sectionID AND_THEN NOT changeRobotsEOAT(robot := robotRight, targetTool := sectionID))
	//NOT (robotLeft.tool = sectionID AND robotRight.tool = sectionID) 
THEN //robots have wrong tool
	//changeRobotsEOAT(robot := robotLeft, targetTool := sectionID); //wait for robots to finish changing tools
	//changeRobotsEOAT(robot := robotRight, targetTool := sectionID);
	RETURN;
END_IF
failLeft := FALSE;
failRight := FALSE;

CASE loadSet OF
	0: //top and bottom
		leftMaterial := pair.top;
		rightMaterial := pair.bottom;
		IF 
			loadingSequenceWB(
				robot:= robotLeft, 
				table:= stagingTableLeft, 
				loadStep:= loadStepLeft, 
				slot:= iSlotLeft,
				suctions:= topSuction,
				surfaceID:= Surface.TOP, 
				material:= pair.top, 
				fail=> failLeft)
			
			AND
			loadingSequenceWB(
				robot:= robotRight,
				table:= stagingTableRight, 
				loadStep:= loadStepRight, 
				slot:= iSlotRight,
				suctions:= bottomSuction,
				surfaceID:= Surface.BOTTOM, 
				material:= pair.bottom, 
				fail=> failRight)
			
		THEN
			loadStepLeft := loadStepRight := 0;
			loadSet := 10;
		END_IF
		
	10: //sides
		leftMaterial := pair.left;
		rightMaterial := pair.right;
		IF
			loadingSequenceWB(
				robot:= robotLeft, 
				table:= stagingTableLeft, 
				loadStep:= loadStepLeft, 
				slot:= iSlotLeft,
				suctions:= leftSuction,
				surfaceID:= Surface.LEFT, 
				material:= pair.left, 
				fail=> )
			
			AND
			loadingSequenceWB(
				robot:= robotRight, 
				table:= stagingTableRight, 
				loadStep:= loadStepRight, 
				slot:= iSlotRight,
				suctions:= rightSuction,
				surfaceID:= Surface.RIGHT, 
				material:= pair.right, 
				fail=> )
			
		THEN
			loadStepLeft := loadStepRight := 0;
			//loadSet := 20;
			loadSet := COMPLETE;
		END_IF
		
	20: //left robot to bottom insertion - module only
		leftMaterial := pair.bottom;
		IF 
			loadingSequenceWB(
				robot:= robotLeft, 
				table:= stagingTableLeft, 
				loadStep:= loadStepLeft, 
				slot:= iSlotLeft,
				suctions:= bottomSuction,
				surfaceID:= Surface.BOTTOM, 
				material:= pair.bottom, 
				fail=> failLeft)
		THEN
			loadSet := COMPLETE;
		END_IF
	
	COMPLETE:
		loadSet := 0;
		loadStepLeft := loadStepRight := 0;
		
		robotLeft.release(sectionID);
		robotRight.release(sectionID);
		
		loadWB := TRUE;
END_CASE
END_METHOD

METHOD splitCombinedMaterials : BOOL
VAR_IN_OUT
	materialID : STRING;
	splitMaterial : STRING;
END_VAR
VAR
	i : INT;
END_VAR
FindAndSplitChar(
	sSeparatorChar:= '_', 
	pSrcString:= ADR(materialID), 
	
	pLeftString:= ADR(splitMaterial), 
	nLeftSize:= SIZEOF(splitMaterial), 
	
	pRightString:= ADR(materialID), 
	nRightSize:= SIZEOF(materialID), 
	
	bSearchFromRight:= FALSE);
END_METHOD

METHOD stage : BOOL
VAR_OUTPUT
	error : BOOL;
END_VAR
sectionID := SectionEnum.WOOD_BUNK;
(*
IF NOT robotLeft.operational OR NOT robotLeft.operational THEN
	error := TRUE;
	RETURN;
END_IF

IF NOT (robotLeft.reserve(reserveRequest := sectionID) AND robotRight.reserve(reserveRequest := sectionID)) THEN
	RETURN;
END_IF

IF NOT (robotLeft.tool = sectionID AND robotRight.tool = sectionID) THEN //robots have wrong tool
	changeRobotsEOAT(robot := robotLeft, targetTool := sectionID); //wait for robots to finish changing tools
	changeRobotsEOAT(robot := robotRight, targetTool := sectionID);
	RETURN;
END_IF
*)

CASE stageSet OF
	0: //create staging template
		IF generateStagingTemplate() THEN
			stageSet := 10;
		END_IF
	
	10: //staging sequence
		IF stagingSequenceLeft(fail => failLeft) AND stagingSequenceRight(fail => failRight)
			(*
			stagingSequence(				
				robot:= robotLeft, 
				commands:= robotLeftOutputs,
				template:= stagingTemplateLeft,
				table:= stagingTableLeft,  
				magazine:= magazineLeft, 
				stagingStep:= stageStepLeft, 
				iSlot:= iSlotLeft,
				fail=> failLeft)
			
			AND
			stagingSequence(
				robot:= robotRight, 
				commands:= robotRightOutputs,
				template:= stagingTemplateRight, 
				magazine:= magazineRight, 
				table:= stagingTableRight, 
				stagingStep:= stageStepRight, 
				iSlot:= iSlotRight,
				fail=> )
			*)
		THEN
			stageStepLeft := stageStepRight := 0;
			iSlotLeft := iSlotRight := 1;
			
			stageSet := COMPLETE;
		END_IF
		
	COMPLETE:
		stagingTemplateRight.clear(); //clear the staging templates
		stagingTemplateLeft.clear();
		
		robotLeft.release(sectionID); //release the robots
		robotRight.release(sectionID);
		
		stageSet := 0;
		stage := TRUE;
		
END_CASE
END_METHOD

METHOD stagingSequenceLeft : BOOL
VAR_OUTPUT
	fail : BOOL;
END_VAR
VAR
	magazineColumn : INT; //valid positions start from 1
END_VAR
VAR CONSTANT
	WIP : INT := 0;
	PASSED : INT := 1;
	FAILED : INT := 2;
	suctionDistance : INT := 15;
END_VAR
IF //staging table is full or matches staging template
	stagingTableLeft.isFull() OR iSlotLeft > 10 OR 
	MEMCMP(ADR(stagingTableLeft.slots), ADR(stagingTemplateLeft.slots), SIZEOF(stagingTableLeft.slots)) = 0
THEN
	stagingSequenceLeft := TRUE;
	RETURN;
END_IF

IF stagingTemplateLeft.slots[iSlotLeft] = '' THEN
	iSlotLeft := iSlotLeft + 1;
	RETURN;
	
ELSIF robotLeft.offline THEN
	fail := TRUE;
	RETURN;
	
ELSIF //robot in used by other section, or has wrong tool and is not done changing
	NOT robotLeft.reserve(reserveRequest := sectionID) OR_ELSE
	(robotLeft.tool <> SectionID AND_THEN NOT changeRobotsEOAT(robot := robotLeft, targetTool := sectionID))
THEN
	RETURN;
END_IF

//follow the stagingTemplateLeft as is
CASE stageStepLeft OF
	0:
		robotLeft.clearCommand();
		
		IF robotLeft.Ready THEN
			stageStepLeft := 10;
		END_IF
		
	10:
		IF NOT magazineLeft.findSlot(materialID := stagingTemplateLeft.slots[iSlotLeft], atSlot => magazineColumn) THEN
			fail := TRUE;
			RETURN;
		END_IF
			
		IF robotLeft.eoatDistance < suctionDistance THEN //robot is grabbing material
			robotLeft.CarryMaterial := magazineLeft.slots[magazineColumn];
		END_IF
		
		IF robotLeft.Done THEN
			stageStepLeft := COMPLETE;
			RETURN;
		ELSIF stagingTableLeft.occupied[iSlotLeft] THEN
			stageStepLeft := 20;
			RETURN;
		END_IF
		
		robotLeft.setGroup(group := 1, value := A21.STAGE_BUNK);
		robotLeft.setGroup(group := 2, value := magazineColumn);
		robotLeft.setGroup(group := 3, value := iSlotLeft);
		
	20:
		IF
			stagingTableLeft.occupied[iSlotLeft] AND //staging table slot is occupied
			stagingTableLeft.slots[iSlotLeft] = '' AND //staging table has not recorded a bunk
			robotLeft.CarryMaterial <> '' //robot is carrying a bunk
		THEN
			stagingTableLeft.place(i := iSlotLeft, materialID := robotLeft.CarryMaterial);
			robotLeft.CarryMaterial := '';
		END_IF
		
		IF robotLeft.Done THEN
			stageStepLeft := COMPLETE;
			RETURN;
		END_IF
		
	COMPLETE:
		(*
		IF stagingTableLeft.occupied[iSlotLeft] THEN //move from gripper to table
			stagingTableLeft.place(i := iSlotLeft, materialID := robotLeft.CarryMaterial);
			robotLeft.CarryMaterial := '';
		END_IF
		*)
		robotLeft.clearCommand();
		
		iSlotLeft := iSlotLeft + 1;
		stageStepLeft := 0;
END_CASE
END_METHOD

METHOD stagingSequenceLeft_old : BOOL
VAR_OUTPUT
	fail : BOOL;
END_VAR
VAR
	magazineColumn : INT; //valid positions start from 1
END_VAR
VAR CONSTANT
	WIP : INT := 0;
	PASSED : INT := 1;
	FAILED : INT := 2;
	suctionDistance : INT := 15;
END_VAR
IF //staging table is full or matches staging template
	stagingTableLeft.isFull() OR iSlotLeft > 10 OR 
	MEMCMP(ADR(stagingTableLeft.slots), ADR(stagingTemplateLeft.slots), SIZEOF(stagingTableLeft.slots)) = 0
THEN
	stagingSequenceLeft_old := TRUE;
	RETURN;
END_IF

IF stagingTemplateLeft.slots[iSlotLeft] = '' THEN
	iSlotLeft := iSlotLeft + 1;
	RETURN;
END_IF

IF //robot in used by other section or has wrong tool
	NOT robotLeft.reserve(reserveRequest := sectionID) OR_ELSE
	(robotLeft.tool <> SectionID AND_THEN changeRobotsEOAT(robot := robotLeft, targetTool := sectionID))
THEN
	RETURN;
END_IF

//follow the stagingTemplateLeft as is
CASE stageStepLeft OF
	0:
		robotLeft.clearCommand();
		MEMSET(ADR(robotLeftOutputs), 0, SIZEOF(robotLeftOutputs));
		
		IF robotLeft.Ready THEN
			stageStepLeft := 10;
		END_IF
		
	10:
		IF NOT magazineLeft.findSlot(materialID := stagingTemplateLeft.slots[iSlotLeft], atSlot => magazineColumn) THEN
			fail := TRUE;
			RETURN;
		END_IF
			
		IF robotLeft.eoatDistance < suctionDistance THEN //robot is grabbing material
			robotLeft.CarryMaterial := magazineLeft.slots[magazineColumn];
		END_IF
		
		IF robotLeft.Done THEN
			stageStepLeft := COMPLETE;
			RETURN;
		END_IF
		
		MEMSET(ADR(robotLeftOutputs), 0, SIZEOF(robotLeftOutputs));
		robotLeft.setGroup(group := 1, value := A21.STAGE_BUNK);
		robotLeft.setGroup(group := 2, value := magazineColumn);
		robotLeft.setGroup(group := 3, value := iSlotLeft);
		robotLeftOutputs[1] := A21.STAGE_BUNK;
		robotLeftOutputs[2] := magazineColumn;
		robotLeftOutputs[3] := iSlotLeft;
		
		robotLeft.setCommand(robotLeftOutputs);
		
	(*
	20:
		
		(*
		MEMSET(ADR(robotLeftOutputs), 0, SIZEOF(robotLeftOutputs));
		robotLeftOutputs[1] := A21.STAGE_BUNK;
		robotLeftOutputs[2] := magazineColumn;
		robotLeftOutputs[3] := iSlotLeft;
		robotLeft.commandEx(robotLeftOutputs);
		*)
		
		robotLeft.commandEx(robotLeftOutputs);
		
		IF stagingTableLeft.occupied[magazineColumn] THEN //move from gripper to table
			stagingTableLeft.place(i := iSlotLeft, materialID := robotLeftMaterial);
			robotLeftMaterial := '';
			stageStepLeft := 30;
		END_IF
				
	30:
		robotLeft.commandEx(robotLeftOutputs);
		IF robotLeft.Done THEN
			stageStepLeft := COMPLETE;
			RETURN;
		END_IF
	*)
	COMPLETE:
		IF stagingTableLeft.occupied[iSlotLeft] THEN //move from gripper to table
			stagingTableLeft.place(i := iSlotLeft, materialID := robotLeft.suspendedMaterial);
			robotLeft.CarryMaterial := '';
		END_IF
		
		
		robotLeft.clearCommand();
		MEMSET(ADR(robotLeftOutputs), 0, SIZEOF(robotLeftOutputs));
		
		iSlotLeft := iSlotLeft + 1;
		stageStepLeft := 0;
END_CASE
END_METHOD

METHOD stagingSequenceRight : BOOL
VAR_OUTPUT
	fail : BOOL;
END_VAR
VAR
	magazineColumn : INT := -1; //valid positions start from 1
END_VAR
VAR CONSTANT
	WIP : INT := 0;
	PASSED : INT := 1;
	FAILED : INT := 2;
	suctionDistance : INT := 15;
END_VAR
IF //staging table is full or matches staging template
	stagingTableRight.isFull() OR iSlotRight > 10 OR 
	MEMCMP(ADR(stagingTableRight.slots), ADR(stagingTemplateRight.slots), SIZEOF(stagingTableRight.slots)) = 0
THEN
	stagingSequenceRight := TRUE;
	RETURN;
END_IF

IF stagingTemplateRight.slots[iSlotRight] = '' THEN
	iSlotRight := iSlotRight + 1;
	RETURN;
	
ELSIF robotRight.offline THEN
	fail := TRUE;
	RETURN;
	
ELSIF //robot in used by other section or has wrong tool
	NOT robotRight.reserve(reserveRequest := sectionID) OR_ELSE
	(robotRight.tool <> SectionID AND_THEN changeRobotsEOAT(robot := robotRight, targetTool := sectionID))
THEN
	RETURN;
END_IF

//follow the stagingTemplateRight as is
CASE stageStepRight OF
	0:
		robotRight.clearCommand();
		
		IF robotRight.Ready THEN
			stageStepRight := 10;
		END_IF
		
	10:
		IF NOT magazineRight.findSlot(materialID := stagingTemplateRight.slots[iSlotRight], atSlot => magazineColumn) THEN
			fail := TRUE;
			RETURN;
		END_IF
			
		IF robotRight.eoatDistance < suctionDistance THEN //robot is grabbing material
			robotRight.CarryMaterial := magazineRight.slots[magazineColumn];
		END_IF
		
		IF robotRight.Done THEN
			stageStepRight := COMPLETE;
			RETURN;
		ELSIF stagingTableRight.occupied[iSlotRight] THEN
			stageStepRight := 20;
			RETURN;
		END_IF
		
		robotRight.setGroup(group := 1, value := A21.STAGE_BUNK);
		robotRight.setGroup(group := 2, value := magazineColumn);
		robotRight.setGroup(group := 3, value := iSlotRight);
		
	20:
		IF
			stagingTableRight.occupied[iSlotRight] AND //staging table slot is occupied
			stagingTableRight.slots[iSlotRight] = '' AND //staging table has not recorded a bunk
			robotRight.CarryMaterial <> '' //robot is carrying a bunk
		THEN
			stagingTableRight.place(i := iSlotRight, materialID := robotRight.CarryMaterial);
			robotRight.CarryMaterial := '';
		END_IF
		
		IF robotRight.Done THEN
			stageStepRight := COMPLETE;
			RETURN;
		END_IF
		
	COMPLETE:
		(*
		IF stagingTableRight.occupied[iSlotRight] THEN //move from gripper to table
			stagingTableRight.place(i := iSlotRight, materialID := robotRight.CarryMaterial);
			robotRight.CarryMaterial := '';
		END_IF
		*)
		robotRight.clearCommand();
		
		iSlotRight := iSlotRight + 1;
		stageStepRight := 0;
END_CASE
END_METHOD

END_PROGRAM

// ---- DUTs/Material Holders/WoodBunkTable.TcPOU
FUNCTION_BLOCK WoodBunkTable EXTENDS MaterialHolder
VAR_OUTPUT
	occupied AT %I* : ARRAY[1..numSlots] OF BOOL; //sensors must turn HIGH before bunk arrives, and turn LOW after bunk leaves
END_VAR
VAR
	i : INT(1..10);
END_VAR
VAR_STAT CONSTANT
	numSlots : INT := 10;
END_VAR

(*
FOR i:=1 TO numSlots BY 1 DO
	IF NOT occupied[i] THEN
		slots[i] := '';
	END_IF
END_FOR
*)

METHOD autofill : BOOL
VAR_INPUT
	materialID : STRING;
END_VAR
VAR
	i : INT;
	slot : INT;
END_VAR
(*
this method will automatically find an open slot
*)
IF isFull() OR materialID = '' THEN
	RETURN;
END_IF

IF findOpenSlot(materialID, openSlot=> slot) THEN
	place(slot, materialID);
	autofill := TRUE;
END_IF
END_METHOD

METHOD findOpenSlot : BOOL
VAR_INPUT
	materialID : STRING;
END_VAR
VAR_OUTPUT
	openSlot : INT := 0;
END_VAR
VAR
	i : INT;
END_VAR
IF FIND(materialID, 'WDW') > 0 THEN //top wide, load in slot 0-1
	FOR i:=1 TO 2 BY 1 DO
		IF slots[i] = '' THEN
			findOpenSlot := TRUE;
			openSlot := i;
			RETURN;
		END_IF
	END_FOR
	
ELSIF FIND(materialID, 'WDT') > 0 OR FIND(materialID, 'WDS') > 0 THEN //top std and sides, load in slot 2-9
	FOR i:=3 TO 10 BY 1 DO
		IF slots[i] = '' THEN
			findOpenSlot := TRUE;
			openSlot := i;
			RETURN;
		END_IF
	END_FOR
	
END_IF
END_METHOD

METHOD findSlot : BOOL
VAR_INPUT
	materialID : STRING;
END_VAR
VAR_OUTPUT
	atSlot : INT;
END_VAR
VAR
	i : INT;
END_VAR
FOR i:=1 TO numSlots BY 1 DO
	IF slots[i] = materialID THEN
		atSlot := i;
		findSlot := TRUE;
		RETURN;
	END_IF
END_FOR
END_METHOD

METHOD isEmpty : BOOL
VAR
	i : INT;
	temp : BOOL;
END_VAR
FOR i:=1 TO numSlots BY 1 DO
	temp := temp OR occupied[i]; //TRUE if any slots are occupied
END_FOR

isEmpty := NOT temp; //invert result - FALSE if any slots are occupied
END_METHOD

METHOD isFull : BOOL
VAR
	i : INT;
	temp : BOOL := TRUE;
END_VAR
FOR i:=1 TO numSlots BY 1 DO
	temp := temp AND occupied[i];
END_FOR

isFull := TEMP;
END_METHOD

METHOD place : BOOL
VAR_INPUT
	i : INT;
	materialID : STRING;
END_VAR
IF slots[i] = '' AND NOT occupied[i] THEN
	slots[i] := materialID;
	place := TRUE;
END_IF
END_METHOD

METHOD remove : BOOL
VAR_INPUT
	i : INT;
END_VAR
VAR_OUTPUT
	materialID : STRING;
END_VAR
IF slots[i] <> '' AND occupied[i] THEN
	materialID := slots[i];
	slots[i] := '';
	
	remove := TRUE;
END_IF
END_METHOD

END_FUNCTION_BLOCK

// ---- DUTs/Material Holders/MaterialHolder.TcPOU
FUNCTION_BLOCK MaterialHolder
VAR_OUTPUT
	slots : ARRAY[1..GVL.maxQueue] OF STRING;
END_VAR

METHOD clear : BOOL
VAR_INPUT
END_VAR
MEMSET(ADR(slots), 0, SIZEOF(slots));
END_METHOD

METHOD findSlot : BOOL
VAR_INPUT
	materialID : STRING;
END_VAR
VAR_OUTPUT
	atSlot : INT := -1;
END_VAR
VAR
	i : INT;
END_VAR
IF materialID = '' THEN
	RETURN;
END_IF

FOR i:=1 TO GVL.maxQueue BY 1 DO
	IF slots[i] = materialID THEN
		atSlot := i;
		findSlot := TRUE;
		RETURN;
	END_IF
END_FOR
END_METHOD

METHOD getSlotsAsArray : POINTER TO STRING
getSlotsAsArray := ADR(slots);
END_METHOD

METHOD setupSlots : BOOL
VAR_INPUT
	setSlots : REFERENCE TO ARRAY[1..GVL.maxQueue] OF STRING;
END_VAR
slots := setSlots;
END_METHOD

END_FUNCTION_BLOCK

// ---- DUTs/Insertion/Insertion.TcPOU
FUNCTION_BLOCK Insertion //2d insertion that combines a slider (alignment) and screw (push)
VAR_INPUT
	enable : BOOL;
END_VAR
VAR_INPUT //interface references to existing drives
	slider : I_EncodedDrive;
	screw : I_ContinuousDrive;
END_VAR
VAR_OUTPUT
	contact AT %I* : BOOL;
	softContact : BOOL; //temporary
	
	busy : BOOL;
	error : BOOL;
	home : BOOL;
	
	homeSet : BOOL;
	
	sliderPos : LREAL;
END_VAR
(*
this FB encapsulates 2 drives into a generic insertion machine
the implementation of both drives should be called externally
an Insertion instance should be called in the scope it is declared in
*)

softContact := slider.contact AND screw.contact; //temporary

homeSet := slider.HomeSet AND screw.HomeSet;

busy := slider.Busy OR screw.Busy;
error := slider.Error OR screw.Error;
home := slider.AtHome AND screw.AtHome;

sliderPos := slider.CurrentPosition;

METHOD align : BOOL
VAR_INPUT
	targetPos : REAL;
END_VAR
slider.moveAbsolute(newTarget := targetPos);
END_METHOD

METHOD homingSequence : BOOL
VAR_INPUT
END_VAR
IF NOT slider.homeSet THEN
	slider.homingSequence();
END_IF

IF NOT screw.homeSet THEN
	screw.homingSequence();
END_IF

homingSequence := homeSet := slider.homeSet AND screw.homeSet;
END_METHOD

METHOD press : BOOL
VAR_INPUT
END_VAR
screw.moveContinuous(direction := MC_Negative_Direction);
END_METHOD

METHOD release : BOOL
VAR_INPUT
END_VAR
screw.moveContinuous(direction := MC_Positive_Direction);
END_METHOD

METHOD traverse : BOOL
VAR_INPUT
	direction : MC_Direction;
END_VAR
slider.moveContinuous(direction := MC_Negative_Direction);
END_METHOD

END_FUNCTION_BLOCK

// ---- POUs/Module Calls/SetupHardware.TcPOU
FUNCTION SetupHardware : BOOL
VAR
	iWoodBunkSlot : WoodBunk;
	iChipboardSlot : Chipboard;
	
	slotsArr : ARRAY[1..GVL.maxQueue] OF STRING;
	
	i : INT;
	j : INT;
	
	temp : INT;
END_VAR

MEMSET(ADR(slotsArr), 0, SIZEOF(slotsArr));
FOR iWoodBunkSlot:=1 TO WoodBunk.size-1 BY 1 DO //init wood bunk magazine slots
	slotsArr[iWoodBunkSlot] := TO_STRING(iWoodBunkSlot);
END_FOR
magazineLeft.setupSlots(slotsArr);
magazineRight.setupSlots(slotsArr);


MEMSET(ADR(slotsArr), 0, SIZEOF(slotsArr));
FOR iChipboardSlot:=1 TO Chipboard.size-1 BY 1 DO //init chipboard skid slots
	slotsArr[iChipboardSlot] := TO_STRING(iChipboardSlot);
END_FOR
skidLeft.setupSlots(slotsArr);
skidRight.setupSlots(slotsArr);


FOR i:=1 TO GVL.maxQueue BY 1 DO //get wood bunk magazine availability from robot
	magazineLeft.setOccupancy(i := i, occupancy := IntegerBitAccess( TO_ULINT(robotLeft.inputs[3]), TO_ULINT(i-1)) );
	skidLeft.setOccupancy(i := i, occupancy := IntegerBitAccess( TO_ULINT(robotLeft.inputs[4]), TO_ULINT(i-1)) );
	
	magazineRight.setOccupancy(i := i, occupancy := IntegerBitAccess( TO_ULINT(robotRight.inputs[3]), TO_ULINT(i-1)) );
	skidRight.setOccupancy(i := i, occupancy := IntegerBitAccess( TO_ULINT(robotRight.inputs[4]), TO_ULINT(i-1)) );
END_FOR

//enable all drives
verticalDriveLeft.bEnable := 
verticalDriveRight.bEnable := 
horizontalDriveLeft.bEnable := 
horizontalDriveRight.bEnable := 
pistonBottom.bEnable := 
TRUE;

END_FUNCTION

// ---- POUs/Module Calls/CallHardwareModules.TcPOU
FUNCTION CallHardwareModules : BOOL //only purpose of this function is to call modules from Hardware
VAR_STAT
	temp : INT;
END_VAR

robotLeft();	
robotRight();

//(*
temp := TO_INT(BoolArrayToInteger(arr := stagingTableLeft.occupied));
temp.15 := NOT strapper.bEnable AND NOT strapper.execute;
robotLeft.setGroup(group := 8, value := temp);

temp := TO_INT(BoolArrayToInteger(arr := stagingTableRight.occupied));
temp.15 := NOT strapper.bEnable AND NOT strapper.execute;
robotRight.setGroup(group := 8, value := temp);
//*)

skidLeft();
skidRight();

stagingTableLeft();
stagingTableRight();

skidLeft();
skidRight();

magazineLeft();
magazineRight();

stagingTableLeft();
stagingTableRight();

strapper();

verticalDriveLeft();
verticalDriveRight();
horizontalDriveLeft();
horizontalDriveRight();
pistonBottom();

END_FUNCTION

// ---- POUs/Utility/BoolArrayToInteger.TcPOU
FUNCTION BoolArrayToInteger : LINT;
VAR_IN_OUT
	arr : ARRAY[*] OF BOOL;
END_VAR
VAR
	i : DINT;
	j : DINT;
END_VAR

BoolArrayToInteger := 0;
(*
FOR i:=LOWER_BOUND(arr, 1) TO UPPER_BOUND(arr, 1) BY 1 DO
	
	IF j < SIZEOF(BoolArrayToInteger) * 8 THEN
		BoolArrayToInteger := SHL(BoolArrayToInteger, 1);
		BoolArrayToInteger.0 := arr[i];
	END_IF
	
END_FOR
*)
//iterate backwards
FOR i:=UPPER_BOUND(arr, 1) TO LOWER_BOUND(arr, 1) BY -1 DO
	
	IF j < SIZEOF(BoolArrayToInteger) * 8 THEN
		BoolArrayToInteger := SHL(BoolArrayToInteger, 1);
		BoolArrayToInteger.0 := arr[i];
	END_IF
	
END_FOR

END_FUNCTION

// ---- DUTs/Machines/RobotA21.TcPOU
FUNCTION_BLOCK RobotA21 EXTENDS KukaRobot
VAR_OUTPUT //from outputs array
	taskID : A21;
	param1 : INT;
	param2 : INT;
	Xmm : INT;
	Ymm : INT;
	Zmm : INT;
	angle : INT;
	stagingOccupancy : INT;
	insertionSuctionStatus : INT;
	magazineStatus : INT; //unused
	inspectionValue : INT;
	
	strapSafetyOut : BOOL;
END_VAR
VAR_OUTPUT //from inputs array
	tool : INT := SectionEnum.WOOD_BUNK;
	suspendedMaterial : STRING;
	//gripper : EOAT := (id := SectionEnum.WOOD_BUNK, material := '');
	
	completedTask : A21;
	eoatDistance : INT;
	magazineAvailability : INT;
	chipboardSkidInPosition : INT;
	materialAtHoldingPosition : INT;
	
	strapSafetyIn : BOOL;
	//robotEOAT : INT; //may not be used
END_VAR

(*
parameters - aliases to IO elements
command - full IO array
*)

SUPER^();

strapSafetyOut := NOT strapper.enable AND NOT strapper.execute;
outputs[8].15 := strapSafetyOut;

outputs[1] := taskID;
outputs[2] := param1;
outputs[3] := param2;
outputs[4] := Xmm;
outputs[5] := Ymm;
outputs[6] := Zmm;
outputs[7] := angle;
outputs[8] := stagingOccupancy;
outputs[9] := insertionSuctionStatus;
outputs[10] := magazineStatus;
outputs[11] := inspectionValue;

outputs[8].15 := strapSafetyOut;

refreshParameters();

{attribute 'monitoring' := 'call'}
PROPERTY Busy : BOOL
GET
VAR
	//emptyOutput : ARRAY[1..50] OF INT;
END_VAR
//Busy stays TRUE until outputs are cleared AND completed task has elapsed
//Ready is always inverse of Busy
refreshParameters();

Busy := taskID <> 0 OR completedTask <> 0;
END_GET
END_PROPERTY

{attribute 'monitoring' := 'call'}
PROPERTY CarryMaterial : STRING
GET
CarryMaterial := suspendedMaterial;
END_GET
SET
suspendedMaterial := CarryMaterial;
END_SET
END_PROPERTY

METHOD clearCommand : BOOL
VAR_INPUT
END_VAR
SUPER^.clearCommand();

refreshParameters();
END_METHOD

{attribute 'monitoring' := 'call'}
PROPERTY Done : BOOL
GET
refreshParameters();

Done :=
	completedTask = taskID AND
	taskID <> 0 AND
	completedTask <> 0;
END_GET
END_PROPERTY

{attribute 'monitoring' := 'call'}
PROPERTY Ready : BOOL
GET
refreshParameters();

Ready := taskID = 0 AND completedTask = 0;
END_GET
END_PROPERTY

METHOD PRIVATE refreshParameters : BOOL
VAR_INPUT
END_VAR
taskID := outputs[1];
param1 := outputs[2];
param2 := outputs[3];
Xmm := outputs[4];
Ymm := outputs[5];
Zmm := outputs[6];
angle := outputs[7];
stagingOccupancy := outputs[8];
insertionSuctionStatus := outputs[9];
magazineStatus := outputs[10]; //unused
inspectionValue := outputs[11];

completedTask := inputs[1];
eoatDistance := inputs[2];
magazineAvailability := inputs[3];
chipboardSkidInPosition := inputs[4];
materialAtHoldingPosition := inputs[5];
//robotEOAT := inputs[6];

strapSafetyIn := inputs[4].15;
END_METHOD

METHOD setCommand : BOOL
VAR_INPUT
	newCommand : REFERENCE TO ARRAY[1..11] OF INT;
END_VAR
MEMCPY(
	ADR(outputs), 
	ADR(newCommand), 
	MIN( SIZEOF(outputs), SIZEOF(newCommand) ));
	
setCommand := Done;

refreshParameters();
END_METHOD

METHOD setGroup : BOOL
VAR_INPUT
	group : INT;
	value : INT;
END_VAR
SUPER^.setGroup(group := group, value := value);

refreshParameters();
END_METHOD

METHOD setParameters : BOOL
VAR_INPUT
	newTaskID : INT;
	newParam1 : INT;
	newParam2 : INT;
	newXmm : INT;
	newYmm : INT;
	newZmm : INT;
	newAngle : INT;
	newStagingOccupancy : INT;
	newInsertionSuctionStatus : INT;
	newMagazineStatus : INT; //unused
	newInspectionValue : INT;
END_VAR
setGroup(group := 1, value := newTaskID);
setGroup(group := 2, value := newParam1);
setGroup(group := 3, value := newParam2);
setGroup(group := 4, value := newXmm);
setGroup(group := 5, value := newYmm);
setGroup(group := 6, value := newZmm);
setGroup(group := 7, value := newAngle);

newStagingOccupancy.15 := NOT strapper.enable AND NOT strapper.execute;
setGroup(group := 8, value := newStagingOccupancy);

setGroup(group := 9, value := newInsertionSuctionStatus);
setGroup(group := 10, value := newMagazineStatus);
setGroup(group := 11, value := newInspectionValue);

refreshParameters();
END_METHOD

END_FUNCTION_BLOCK

// ---- DUTs/Machines/KukaRobot.TcPOU
FUNCTION_BLOCK KukaRobot
VAR_OUTPUT
	forceStop AT %Q* : BOOL;
	resetSignal AT %Q* : BOOL;
	
	outputs AT %Q* : ARRAY[1..50] OF INT;
	inputs AT %I* : ARRAY[1..20] OF INT;
	
	taskID : INT;
	completedTask : INT;
	
	operational : BOOL;
	reserved : BOOL;
	reservation : SectionEnum := SectionEnum.NULL_SECTION;
	tool : SectionEnum := SectionEnum.WOOD_BUNK;
	
	error : BOOL;
	errId : DINT;
END_VAR
VAR
	step : (SEND_COMMAND, WAIT);
END_VAR

taskID := outputs[1];
completedTask := inputs[1];

{attribute 'monitoring' := 'variable'}
{attribute 'monitoring' := 'call'}
PROPERTY Busy : BOOL
GET
VAR
	emptyOutput : ARRAY[1..50] OF INT;
END_VAR

//Busy stays TRUE until outputs are cleared AND completed task has elapsed
//Ready is always inverse of Busy
updateStatus();

Busy :=
	MEMCMP(ADR(outputs), ADR(emptyOutput), SIZEOF(outputs)) <> 0 OR
	completedTask <> 0;
END_GET
END_PROPERTY

METHOD commandEx : BOOL
VAR_INPUT
	newOutputs : REFERENCE TO ARRAY[1..50] OF INT;
END_VAR
outputs := newOutputs;
END_METHOD

//{attribute 'monitoring' := 'variable'}
{attribute 'monitoring' := 'call'}
PROPERTY Done : BOOL
GET
updateStatus();

Done := completedTask = taskID;
END_GET
END_PROPERTY

METHOD eStop : BOOL
VAR_INPUT
END_VAR
forceStop := TRUE;
eStop := TRUE;
END_METHOD

METHOD idleCommand : BOOL
VAR_INPUT
END_VAR
MEMSET(ADR(outputs), 0, SIZEOF(outputs));
END_METHOD

PROPERTY Ready : BOOL
GET
updateStatus();

Ready := NOT Busy;
END_GET
END_PROPERTY

METHOD release : BOOL
VAR_INPUT
	sectionReservation : SectionEnum;
END_VAR
IF reservation = sectionReservation AND reserved THEN
	reservation := SectionEnum.NULL_SECTION;
	reserved := FALSE;
	release := TRUE;
END_IF
END_METHOD

METHOD reserve : BOOL
VAR_INPUT
	reserveRequest : SectionEnum;
END_VAR
(*
this method exists because chipboard and wood bunk operations use the same robot
both sections need to check if the robot is open to commands before use
*)
IF reserved AND reservation = reserveRequest THEN
	reserve := TRUE;

ELSIF (NOT reserved) AND reservation = SectionEnum.NULL_SECTION THEN
	reservation := reserveRequest;
	reserved := TRUE;
	reserve := TRUE;

END_IF
END_METHOD

METHOD reset : BOOL
//resetSignal := TRUE;
//done := FALSE;

MEMSET(ADR(outputs), 0, SIZEOF(outputs));
(*
IF ready AND completedTask = 0 THEN
	resetSignal := FALSE;
	reset := TRUE;
END_IF
*)
END_METHOD

METHOD resume : BOOL
VAR_INPUT
END_VAR
forceStop := FALSE;

resume := NOT error AND errId = 0;
END_METHOD

METHOD setCommandAndWait : BOOL
VAR_INPUT
	newOutputs : REFERENCE TO ARRAY[1..50] OF INT;
END_VAR
//IF NOT Busy THEN
	//RETURN;
//END_IF

outputs := newOutputs;
setCommandAndWait := Done;

(*
CASE step OF
	SEND_COMMAND: //wait 1 cycle
		outputs := newOutputs;
		step := WAIT;
		
	WAIT:
		IF done THEN
			(*	
			IF NOT reset() THEN
				RETURN;
			END_IF
			
			step := 0;
			*)
			setCommandAndWait := TRUE;
		END_IF
		
END_CASE
*)
END_METHOD

METHOD updateStatus : BOOL
VAR_INPUT
END_VAR
taskID := outputs[1];
completedTask := inputs[1];
END_METHOD

END_FUNCTION_BLOCK

// ---- POUs/Utility/String Array/AddToStringArray.TcPOU
FUNCTION AddToStringArray : BOOL
VAR_IN_OUT
	arr : ARRAY[*] OF STRING; //must start from 0 index
END_VAR
VAR_INPUT
	newString : STRING;
END_VAR
VAR_OUTPUT
	numElements : DINT;
	nextIndex : DINT;
END_VAR
VAR
	i : DINT;
END_VAR

FOR i:=LOWER_BOUND(arr, 1) TO UPPER_BOUND(arr, 1) BY 1 DO
	numElements := numElements + 1;
	
	IF arr[i] = '' THEN
		
		arr[i] := newString;
		nextIndex := i + 1;
		
		AddToStringArray := TRUE;
		EXIT;
	END_IF
END_FOR

END_FUNCTION

// ---- DUTs/Material Holders/SkidMagazine.TcPOU
FUNCTION_BLOCK SkidMagazine EXTENDS MaterialHolder
VAR_OUTPUT
	occupied : ARRAY[1..GVL.maxQueue] OF BOOL;
	
	inPosition1 AT %I* : BOOL;
	inPosition2 AT %I* : BOOL;
END_VAR

METHOD setOccupancy : BOOL
VAR_INPUT
	i : INT;
	occupancy : BOOL;
END_VAR
occupied[i] := occupancy;
END_METHOD

END_FUNCTION_BLOCK

// ---- DUTs/Machines/StrapMachine.TcPOU
FUNCTION_BLOCK StrapMachine
VAR_INPUT
	bEnable : BOOL;
END_VAR
VAR_OUTPUT
	enable AT %Q* : BOOL;
	error AT %I* : BOOL;
	ready AT %I* : BOOL;
	//busy (*AT %I**) : BOOL;
	done AT %I* : BOOL;
	home AT %I* : BOOL;
	
	execute AT %Q* : BOOL;
	reset AT %Q* : BOOL;
	
	timeout : BOOL;
	
	atBundleLevel AT %I* : BOOL;
END_VAR
VAR	
	holdPost : TON;
	delay : TON;
	
	start : BOOL;
	step : (SETUP, RUN, WAIT);
END_VAR
VAR_STAT CONSTANT
	pulseTime : TIME := T#100MS;
	holdTime : TIME := T#500MS;
	maxDelay : TIME := T#30S;
END_VAR

holdPost(IN:= , PT:= holdTime, Q=> , ET=> );
delay(IN:= step > 0 OR start, PT:= maxDelay, Q=> timeout, ET=> );

IF delay.Q THEN
	delay.IN := FALSE;
	//timeout := TRUE;
	//busy := FALSE;
	
	start := FALSE;
	step := SETUP;
END_IF

CASE step OF
	SETUP:
		//busy := FALSE;
		enable := FALSE;
		execute := FALSE;
		
		IF NOT clear() THEN
			RETURN;
		END_IF		
		
		enable := bEnable AND robotLeft.strapSafetyIn AND robotRight.strapSafetyIn;
		
		IF start AND enable THEN
			start := FALSE;
			step := RUN;
		END_IF
	
	RUN:
		IF NOT execute THEN
			execute := TRUE;
			RETURN; //keeps execute TRUE for at least 1 cycle
		END_IF
		
		IF execute AND NOT ready AND NOT home THEN
			execute := FALSE;
			step := WAIT;
		END_IF
		
	WAIT:
		IF home THEN
			holdPost.IN := TRUE;
			enable := FALSE;
			execute := FALSE;
		END_IF
		
		IF holdPost.Q THEN
			holdPost.IN := FALSE;
			done := TRUE;
			step := 0;
		END_IF
		
END_CASE

(*
executePulse(IN:= , PT:= pulseTime, Q=> , ET=> );
execute := executePulse.IN AND NOT executePulse.Q;

IF executePulse.Q THEN
	executePulse.IN := FALSE;
END_IF


resetPulse(IN:= , PT:= pulseTime, Q=> , ET=> );
StrapMachineST.reset := resetPulse.IN AND NOT resetPulse.Q;

IF resetPulse.Q THEN
	executePulse.IN := FALSE;
END_IF

ready := enable AND NOT execute AND NOT StrapMachineST.reset AND NOT error AND home;
*)

METHOD clear : BOOL
VAR_INPUT
END_VAR
(*
reset should be continuously called until machine returns evidence that it is ready again
machine is expected to not respond to reset signals if it is already in an idle state
*)
enable := FALSE;
execute := FALSE;

IF error THEN
	reset := NOT reset;
ELSE
	reset := FALSE;
END_IF

clear := NOT error;
END_METHOD

METHOD strap : BOOL
VAR_INPUT
END_VAR
//IF ready AND NOT busy AND NOT error THEN
	//busy := TRUE;
	//start := TRUE;
	//strap := TRUE;
//END_IF

start := TRUE;
END_METHOD

END_FUNCTION_BLOCK

// ---- DUTs/Insertion/Drives/ClearLinkMC.TcPOU
FUNCTION_BLOCK ClearLinkMC EXTENDS FBA_Drive IMPLEMENTS I_EncodedDrive //I_PositionalDrive, I_ContinuousDrive
VAR_OUTPUT
	pulse AT %Q* : INT; //num pulses
	outputRegister AT %Q* : INT;
	brakeRelease AT %Q* : BOOL;
	
	A : BOOL; //direction (F = inwards, T = outwards)
	B : BOOL; //home bit
	clear : BOOL;
	
	hlfb AT %I* : REAL; //high level feedback, if -9999 then servo is idle
	position, targetPos : LREAL;
END_VAR
VAR
	pulseRequest : INT;
	
	minHoming : TON;
	resetTimer : TP;
	
	mode : (DISABLE, HOLD, TARGET, CONTINUOUS, RESET_ERR);
END_VAR
VAR_STAT CONSTANT
	resetTime : TIME := T#1000MS;
	unitsPerPulse : INT := 800; //800 Teknic units per revolution
	distancePerPulse : INT := 5; //5mm per revolution
END_VAR

//M-connector output register
outputRegister.0 := bEnable; 	//enable
outputRegister.1 := A; 			//direction bit
outputRegister.2 := B; 			//homing bit - set to TRUE after startup to begin homing, then set to FALSE to finish homing
outputRegister.3 := clear; 		//reset bit

resetTimer(IN:= , PT:= resetTime, Q=> clear, ET=> ); //reset timer

IF NOT bEnable THEN
	homingComplete := FALSE;
	mode := HOLD;
END_IF

override(); //if sensor limits are reached, this method blocks motion that would exceed the limits

CASE mode OF		
	HOLD: //hold current position, no motion
		pulse := 0;
		pulseRequest := 0;
	
	TARGET:	//target a given position
		IF WithinTolerance(position, targetPos, distancePerPulse) THEN
			pulseRequest := 0;
			mode := HOLD;
			
		ELSIF NOT Busy THEN
			A :=  position < targetPos;
			(*
			2 options to traverse to a target position:
				a)  send all pulses at once - single continuous motion but may exceed limits
				b)  1 pulse at a time - choppy but safer
			*)
			//pulseRequest := TO_INT(ABS(position - targetPos)/distancePerPulse);
			pulseRequest := 1;
			
		END_IF
		
	CONTINUOUS: //single pulses in the direction specified by moveContinuous()
		pulseRequest := 1;
		
	RESET_ERR: //reset pulse, servo may need to be rehomed aftewards
		pulse := 0;
		pulseRequest := 0;
		resetTimer.IN := TRUE;
		
		IF resetTimer.Q THEN
			resetTimer.IN := FALSE;
			mode := HOLD;
		END_IF
		
END_CASE

sequence();

PROPERTY Busy : BOOL
GET
Busy := hlfb <> -9999;
END_GET
END_PROPERTY

PROPERTY CurrentPosition : LREAL
GET
CurrentPosition := position;
END_GET
SET
position := CurrentPosition;
END_SET
END_PROPERTY

PROPERTY Error : BOOL
GET
END_GET
END_PROPERTY

METHOD homingSequence : BOOL
minHoming(IN:= , PT:= T#1S, Q=> , ET=> ); //IN and OUT should be held for at least 1 second - may be removed for deployment

IF NOT bEnable THEN //homing does not begin until software enable
	RETURN;
END_IF

CASE step OF
	Homing.IDLE:
		bEnable := FALSE;
		A := FALSE;
		B := FALSE;
		brakeRelease := TRUE;
		
		homingComplete := FALSE;
		step := Homing.IN;
		
	Homing.IN: //let insertion drop to inner limit before homing
		bEnable := FALSE;
		A := FALSE;
		B := FALSE;
		brakeRelease := TRUE;
		
		minHoming.IN := TRUE;
		
		IF NOT innerLimit AND minHoming.Q THEN
			minHoming.IN := FALSE;
			step := Homing.OUT;
		END_IF
	
	Homing.OUT:
		bEnable := TRUE;
		A := FALSE;
		B := TRUE;
		brakeRelease := TRUE;
		
		minHoming.IN := TRUE;
		
		IF NOT home AND minHoming.Q THEN
			minHoming.IN := FALSE;
			step := Homing.DONE;
		END_IF
		
	Homing.DONE:
		bEnable := TRUE;
		A := FALSE;
		B := FALSE;
		brakeRelease := TRUE;
			
		position := 0;
		
		homingComplete := TRUE;
		homingSequence := TRUE;
		
		mode := HOLD;
		step := Homing.IDLE;
	
END_CASE
END_METHOD

METHOD moveAbsolute : BOOL
VAR_INPUT
	newTarget : LREAL;
END_VAR
targetPos := newTarget;
mode := TARGET;
END_METHOD

METHOD moveContinuous : BOOL
VAR_INPUT
	direction : MC_Direction;
END_VAR
IF direction = MC_Negative_Direction THEN
	A := FALSE;
ELSIF direction = MC_Positive_Direction THEN
	A := TRUE;
END_IF

mode := CONTINUOUS;
END_METHOD

METHOD moveRelative : BOOL
VAR_INPUT
	distance : LREAL;
END_VAR
targetPos := targetPos + distance;

mode := TARGET;
END_METHOD

METHOD PRIVATE override : BOOL
VAR_INPUT
END_VAR
(*
IF (*NOT*) home THEN //block outwards motion
	position := 0;
	IF A THEN
		mode := HOLD;
	END_IF
	
ELSIF (*NOT*) outerLimit AND_THEN A THEN //block outwards motion
	mode := HOLD;

ELSIF (*NOT*) innerLimit AND_THEN NOT A THEN //block inwards motion
	mode := HOLD;
	
END_IF
*)


IF
	((*NOT*) home AND_THEN A) OR
	((*NOT*) outerLimit AND_THEN A) OR
	((*NOT*) innerLimit AND_THEN NOT A)
THEN
	mode := HOLD;
END_IF


IF (*NOT*) home THEN //block outwards motion
	position := 0;
END_IF
END_METHOD

METHOD reset : BOOL
VAR_INPUT
END_VAR
mode := RESET_ERR;
END_METHOD

METHOD PRIVATE sequence : BOOL
VAR_INPUT
END_VAR
IF Busy THEN //servo is active
	IF A THEN //positive direction
		position := position + (distancePerPulse * pulse);
	ELSE //negative direction
		position := position - (distancePerPulse * pulse);
	END_IF
	pulse := 0; //pulses already received, can be set to 0 so position change is not compounded

ELSIF pulse = 0 THEN //servo is not active
	pulse := pulseRequest;
	pulseRequest := 0; //remove this if not working as intended
	
END_IF
END_METHOD

METHOD stop : BOOL
VAR_INPUT
END_VAR
mode := HOLD;
END_METHOD

PROPERTY TargetPosition : LREAL
GET
END_GET
SET
targetPos := TargetPosition;
END_SET
END_PROPERTY

END_FUNCTION_BLOCK

// ---- DUTs/Insertion/Prototypes/FBA_Drive.TcPOU
FUNCTION_BLOCK ABSTRACT FBA_Drive IMPLEMENTS I_Drive
VAR_INPUT
	bEnable : BOOL;
END_VAR
VAR_OUTPUT
	contactSensor AT %I* : BOOL;
	
	outerLimit AT %I* : BOOL;
	home AT %I* : BOOL;
	innerLimit AT %I* : BOOL;
	(*
	busy : BOOL;
	contact : BOOL;
	error : BOOL;
	homeSet : BOOL;
	*)
	homingComplete : BOOL;
END_VAR
VAR
	step : Homing;
END_VAR
(*
this abstract FB only contains the bare minimum types for any drive/servo
*)

PROPERTY AtHome : BOOL
GET
AtHome := home;
END_GET
END_PROPERTY

PROPERTY AtInnerLimit : BOOL
GET
AtInnerLimit := innerLimit;
END_GET
END_PROPERTY

PROPERTY AtOuterLimit : BOOL
GET
AtOuterLimit := outerLimit;
END_GET
END_PROPERTY

PROPERTY ABSTRACT Busy : BOOL
GET
END_GET
END_PROPERTY

PROPERTY Contact : BOOL
GET
Contact := contactSensor;
END_GET
END_PROPERTY

PROPERTY ABSTRACT Error : BOOL
GET
END_GET
END_PROPERTY

PROPERTY HomeSet : BOOL
GET
HomeSet := homingComplete;
END_GET
END_PROPERTY

METHOD ABSTRACT homingSequence : BOOL
VAR_INPUT
END_VAR
END_METHOD

METHOD ABSTRACT stop : BOOL
VAR_INPUT
END_VAR
END_METHOD

END_FUNCTION_BLOCK
